Staubli VAL3: num2bool.pgx

public program num2bool(num& x_nInput[], bool& x_bResult[], bool& x_bError)
  local num l_nLength
  local num l_nElement
begin

  x_bError = false
  l_nLength = size(x_nInput)
  x_bResult = false
  resize(x_bResult, 1,l_nLength)

  for l_nElement = 0 to l_nLength-1
    if x_nInput[l_nElement] == 0
      x_bResult[l_nElement] = false
    elseIf x_nInput[l_nElement] == 1
      x_bResult[l_nElement] = true
    else
      x_bError = true
    endIf
  endFor

end
